Staubli VAL3: getFrame.pgx

public program getFrame(frame& x_fFrame[], bool x_bCycle)
begin
  if x_bCycle
    x_fFrame.trsf=position(pt:tTraj[sItemCycle].fFrame,world)
  else
    // update the frame
    x_fFrame.trsf=position(pEditPoint.fFrame,world)
  endIf
end
